(*Basic MAIN with an example organiser and scam*)
{info '_Welcome to the Boikon Twincat 3 Template'}
{info '__Please read the _Readme.txt for more info'}
{warning 'TODO Template: upload boot project at online change is disabled in project settings, RE-ENABLE!!!!'}
PROGRAM MAIN
VAR
	//General collection of system wide IO and control blocks
	General: Utl_General;

	//TODO TEMPLATE: here in the example only 1 organiser is used, add + rename as needed
	Organiser:cntrl_Organiser(						
		SP_TmrReset := T#1S,
		SP_TmrResetES := T#3S);
END_VAR

//TODO TEMPLATE >> Remove this section, it is for testing the library and template
//Also remove the define from here: project/properties/compile/compiler defines/IsTemplate
{IF defined (IsTemplate)}
	{warning 'TODO Template: testing is enabled >> Remove the define and clean all "TODO TEMPLATE" locations'}
	{attribute 'analysis' := '-33'}
	VAR
		//Scam-template >> use tool supplied in the folder, to make a copy for your own scam implementation 
		OrganiserFake: cntrl_OrganiserFake;
		
		//Fully functional test scam which uses almost all library blocks >> can be used as example how to do things 
		ExampleMachinePart: SCM_TemplateClean;

		//just to show it's possible
		//these variables will now have the same comment (these 2 lines)
		//*multiline comment still is a kind of broken in the editor, parts will dissapear..
		MyBool1,MyBool2,MyBool3:BOOL;  

		//Banner-Multicolor signal lamp
		//NOTE: You can use it this way for multiple organisers as well, just keep calling ..M_UpdateOrganiserState(xxx) for each organiser  
		LP_OrgGroupMachinePart:Cntrl_BannerKxx(
			Intensity:= eBannerKxx_Intensity.Low);

		LP_MurrTest: cntrl_MurrModLight60(NrOfStacks:=3);

		//Performance test	
		HM_ProfileBlocks:BOOL;
		StopWatchGeneral,StopWatchMachineStuff:profiler;
		
		//casting works with a lot of types, example time
		sMyUtcTime:string;

		//string value to int test
		sValue1,sValue2,sValue3:STRING := '123';
		sValue4,sValue5:string(1);
		b0Value:BYTE;
		iValue1,iValue2:INT;
		
		
		//random tests
		dbglreal:LREAL;
		dbgbool1,dbgbool2,dbgbool3:BOOL;
	END_VAR
{END_IF}

//TODO template: general actions can be added here. 
//in utl_General I've added the usual suspects needed for a machine.
//please keep in mind I've only included common reocurring items, you need to thoroughly check / update / clean the block!
a_General();
b_MachinePart();

ACTION a_General:
//General is the place for all in-/outputs not specific belonging to a machinepart like:
//	-handling of boikonlibrary functionality
//	-general start/stop/reset buttons + lights
//	-general airpressure sensor
//	-safety components: control + errors for doors/lightscreens/pushbuttons
//	-ethercat diagnostics
General(
	//Reset command + general start/stop/reset button lights > add organisers as needed, use OR
	I_SN_ResetErrors:= Organiser.Reset_K,
	I_SN_Lp_Pb_StartAll:= Organiser.Q_LP_Start,
	I_SN_Lp_Pb_StopAll:= Organiser.Q_LP_Stop,
	I_SN_Lp_Pb_ResetAll:= Organiser.Q_LP_Reset,
	
	//Machine status
	I_STS_Error:=,
	I_STS_NoDischarge:=,
	I_STS_OperatorInput:=,
	I_STS_Running:=,	
	
	//Organiser/SCAM control-outputs
	Q_SN_ES_Zone1_OK=>, 
	Q_SN_StartAll=>,
	Q_SN_StopAll=>,
	Q_SN_ResetAll=> ,
	Q_SN_TotalResetAll=>);

//TODO TEMPLATE remove if not needed
//Organiser(s) Banner multicolor indicator light
//	this is an example on how to use it to show the status of an organiser
//	1) you can also manually control the lamp with the given M_Set... methods, but then don't call M_UpdateOrganiserState anymore!
//	2) inside general would be a better place but there you can't access the Organiser instances easily (or you tresspass OOP by doing things like: main.Organiser inside.... > don't do that!)
LP_OrgGroupMachinePart.M_UpdateOrganiserState(Organiser); //call this method for each organiser belonging to this group
LP_OrgGroupMachinePart();

//TODO TEMPLATE remove banner break-time
//Mess around with the banner multicolor lamp >> if break-time, overwrite previous (organiser-state) call with a manual set color
IF(	(	BknGlbl.LocalSystemTime.wHour = 10
		AND_THEN BknGlbl.LocalSystemTime.wMinute <= 15)
	OR	(	BknGlbl.LocalSystemTime.wHour = 12
			AND_THEN BknGlbl.LocalSystemTime.wMinute >= 30)
	OR	(	BknGlbl.LocalSystemTime.wHour >= 17))
THEN
	LP_OrgGroupMachinePart.M_Set2ColorAnimation(
		I_Color1 := eBannerKxx_Color.Yellow,
		I_Color2 := eBannerKxx_Color.Red,
		I_Animation:= eBannerKxx_AnimationType.HalfHalfRotate,
		TRUE); 
	LP_OrgGroupMachinePart();
END_IF
END_ACTION

ACTION b_MachinePart:
//Note: if the machine consists of several machine parts with their own organiser then for a cleaner structure make a seperate action for each part
//todo think about this

Organiser(
	//Emergencystop zone for scams connected to this organiser
	I_SN_ES_OK:= General.Q_SN_ES_Zone1_OK,
	I_SN_ExternalError:= General.Q_SN_ERR_General, //organiser should go into error caused by external factors (like a general error)
	//Total reset command for this organiser and connected scams
	//note: scams that communicate with each other via interlocking should have the same total reset command otherwise deadlocks will occur!
	I_SN_TotalReset:= General.Q_SN_TotalResetAll,
	I_PB_Start:= General.Q_SN_StartAll,
	I_PB_Stop:= General.Q_SN_StopAll,
	I_PB_Reset:= General.Q_SN_ResetAll, 
	Q_LP_Start=>, 
	Q_LP_Stop=>, 
	Q_LP_Reset=>);

ExampleMachinePart( //todo remove true
	I_K_ES_OK:= General.Q_SN_ES_Zone1_OK, 			//Emergency stop for this zone OK. @ mutliple zones, fbGeneral must be adapted to supply these signals for each zone
	I_Organiser:= Organiser, 						//Control signals from the organiser
	I_STS_SUP_Empty:= , 							//Connect to upstream. The upstream is empty, use this to enter energy-save mode (stop conveyors etc)
	Q_STS_Empty=> , 								//Connect to downstream. The supply is empty and this part is now empty and in energy-save mode
	Q_SN_SUP_Request=> ,							//Connect to upstream. This program is running and ready to receive products
);
END_ACTION

END_PROGRAM

(* stored: Version 1.1.0.1
   POU MAIN: Id {55a103d2-858d-4dc1-a31e-5fbbbfc40857}, SpecialFunc None
   Action a_General: Id {ef997c49-6f4c-4175-83bc-febdc880087c}
   Action b_MachinePart: Id {51166692-ba41-42d3-9f46-75bf2fc7547e} *)
